FUNCTION_BLOCK PAEActValve_3pos EXTENDS PAEActuator1way_3pos
VAR_INPUT
END_VAR
VAR_OUTPUT
END_VAR
VAR
END_VAR

METHOD PUBLIC PAEActValve_3pos
VAR_INPUT
END_VAR
END_METHOD

END_FUNCTION_BLOCK

(* stored: Version 1.1.0.1, ProductVersion 3.1.4020.12
   POU PAEActValve_3pos: Id {eb3052ef-90bd-4b86-8aa5-b004af49add2}, SpecialFunc None
   Method PAEActValve_3pos: Id {b3719bdf-5bd1-498f-8466-22ba5f5fb939} *)
